// TwinCAT 3 PLC project Untitled1
// ProgramVersion: 3.1.4026.15
// libraries:
//   Tc2_Standard, * (Beckhoff Automation GmbH)
//   Tc2_System, * (Beckhoff Automation GmbH)
//   Tc2_TcpIp, * (Beckhoff Automation GmbH)
// project tree:
//   DUTs/ E_TcpIpErrorID.TcDUT, E_TcpIpState.TcDUT
//   / PlcTask.TcTTO
//   POUs/ FB_TCPIPServerManager.TcPOU, FB_TCPIPClientManager.TcPOU, MAIN.TcPOU
// real-time tasks:
//   TASK PlcTask: cycle T#10ms, priority 20, ADS port 350

CONFIGURATION Untitled1
    RESOURCE PLC ON TwinCAT3
        TASK PlcTask(INTERVAL := T#10ms, PRIORITY := 20);
        PROGRAM MAIN WITH PlcTask : MAIN;
    END_RESOURCE
END_CONFIGURATION

// ---- DUTs/E_TcpIpErrorID.TcDUT
{attribute 'qualified_only'}
//{attribute 'strict'}
{attribute 'to_string'}
TYPE E_TcpIpErrorID :
(
	ERR_NOERROR := 0,
	ERR_INTERNAL := 1,
	ERR_NORTIME := 2,
	ERR_ALLOCLOCKEDMEM := 3,
	ERR_INSERTMAILBOX := 4,
	ERR_WRONGRECEIVEHMSG := 5,
	ERR_TARGETPORTNOTFOUND := 6,
	ERR_TARGETMACHINENOTFOUND := 7,
	ERR_UNKNOWNCMDID := 8,
	ERR_BADTASKID := 9,
	ERR_NOIO := 10,
	ERR_UNKNOWNAMSCMD := 11,
	ERR_WIN32ERROR := 12,
	ERR_PORTNOTCONNECTED := 13,
	ERR_INVALIDAMSLENGTH := 14,
	ERR_INVALIDAMSNETID := 15,
	ERR_LOWINSTLEVEL := 16,
	ERR_NODEBUGINTAVAILABLE := 17,
	ERR_PORTDISABLED := 18,
	ERR_PORTALREADYCONNECTED := 19,
	ERR_AMSSYNC_W32ERROR := 20,
	ERR_AMSSYNC_TIMEOUT := 21,
	ERR_AMSSYNC_AMSERROR := 22,
	ERR_AMSSYNC_NOINDEXINMAP := 23,
	ERR_INVALIDAMSPORT := 24,
	ERR_NOMEMORY := 25,
	ERR_TCPSEND := 26,
	ERR_HOSTUNREACHABLE := 27,
	ERR_INVALIDAMSFRAGMENT := 28,
	ERR_TLSSEND := 29,
	ERR_ACCESSDENIED := 30,

	(* Router error codes *)
	ROUTERERR_NOLOCKEDMEMORY := 1280,
	ROUTERERR_RESIZEMEMORY := 1281,
	ROUTERERR_MAILBOXFULL := 1282,
	ROUTERERR_DEBUGBOXFULL := 1283,
	ROUTERERR_UNKNOWNPORTTYPE := 1284,
	ROUTERERR_NOTINITIALIZED := 1285,
	ROUTERERR_PORTALREADYINUSE := 1286,
	ROUTERERR_NOTREGISTERED := 1287,
	ROUTERERR_NOMOREQUEUES := 1288,
	ROUTERERR_INVALIDPORT := 1289,
	ROUTERERR_NOTACTIVATED := 1290,
	ROUTERERR_FRAGMENTBOXFULL := 1291,
	ROUTERERR_FRAGMENTTIMEOUT := 1292,
	ROUTERERR_TOBEREMOVED := 1293,

	(* General ADS error codes *)
	ADSERR_DEVICE_ERROR := 1792,
	ADSERR_DEVICE_SRVNOTSUPP := 1793,
	ADSERR_DEVICE_INVALIDGRP := 1794,
	ADSERR_DEVICE_INVALIDOFFSET := 1795,
	ADSERR_DEVICE_INVALIDACCESS := 1796,
	ADSERR_DEVICE_INVALIDSIZE := 1797,
	ADSERR_DEVICE_INVALIDDATA := 1798,
	ADSERR_DEVICE_NOTREADY := 1799,
	ADSERR_DEVICE_BUSY := 1800,
	ADSERR_DEVICE_INVALIDCONTEXT := 1801,
	ADSERR_DEVICE_NOMEMORY := 1802,
	ADSERR_DEVICE_INVALIDPARM := 1803,
	ADSERR_DEVICE_NOTFOUND := 1804,
	ADSERR_DEVICE_SYNTAX := 1805,
	ADSERR_DEVICE_INCOMPATIBLE := 1806,
	ADSERR_DEVICE_EXISTS := 1807,
	ADSERR_DEVICE_SYMBOLNOTFOUND := 1808,
	ADSERR_DEVICE_SYMBOLVERSIONINVALID := 1809,
	ADSERR_DEVICE_INVALIDSTATE := 1810,
	ADSERR_DEVICE_TRANSMODENOTSUPP := 1811,
	ADSERR_DEVICE_NOTIFYHNDINVALID := 1812,
	ADSERR_DEVICE_CLIENTUNKNOWN := 1813,
	ADSERR_DEVICE_NOMOREHDLS := 1814,
	ADSERR_DEVICE_INVALIDWATCHSIZE := 1815,
	ADSERR_DEVICE_NOTINIT := 1816,
	ADSERR_DEVICE_TIMEOUT := 1817,
	ADSERR_DEVICE_NOINTERFACE := 1818,
	ADSERR_DEVICE_INVALIDINTERFACE := 1819,
	ADSERR_DEVICE_INVALIDCLSID := 1820,
	ADSERR_DEVICE_INVALIDOBJID := 1821,
	ADSERR_DEVICE_PENDING := 1822,
	ADSERR_DEVICE_ABORTED := 1823,
	ADSERR_DEVICE_WARNING := 1824,
	ADSERR_DEVICE_INVALIDARRAYIDX := 1825,
	ADSERR_DEVICE_SYMBOLNOTACTIVE := 1826,
	ADSERR_DEVICE_ACCESSDENIED := 1827,
	ADSERR_DEVICE_LICENSENOTFOUND := 1828,
	ADSERR_DEVICE_LICENSEEXPIRED := 1829,
	ADSERR_DEVICE_LICENSEEXCEEDED := 1830,
	ADSERR_DEVICE_LICENSEINVALID := 1831,
	ADSERR_DEVICE_LICENSESYSTEMID := 1832,
	ADSERR_DEVICE_LICENSENOTIMELIMIT := 1833,
	ADSERR_DEVICE_LICENSEFUTUREISSUE := 1834,
	ADSERR_DEVICE_LICENSETIMETOLONG := 1835,
	ADSERR_DEVICE_EXCEPTION := 1836,
	ADSERR_DEVICE_LICENSEDUPLICATED := 1837,
	ADSERR_DEVICE_SIGNATUREINVALID := 1838,
	ADSERR_DEVICE_CERTIFICATEINVALID := 1839,
	ADSERR_DEVICE_LICENSEOEMNOTFOUND := 1840,
	ADSERR_DEVICE_LICENSERESTRICTED := 1841,
	ADSERR_DEVICE_LICENSEDEMODENIED := 1842,
	ADSERR_DEVICE_INVALIDFNCID := 1843,
	ADSERR_DEVICE_OUTOFRANGE := 1844,
	ADSERR_DEVICE_INVALIDALIGNMENT := 1845,
	ADSERR_DEVICE_LICENSEPLATFORM := 1846,
	ADSERR_DEVICE_FORWARD_PL := 1847,
	ADSERR_DEVICE_FORWARD_DL := 1848,
	ADSERR_DEVICE_FORWARD_RT := 1849,
	ADSERR_CLIENT_ERROR := 1856,
	ADSERR_CLIENT_INVALIDPARM := 1857,
	ADSERR_CLIENT_LISTEMPTY := 1858,
	ADSERR_CLIENT_VARUSED := 1859,
	ADSERR_CLIENT_DUPLINVOKEID := 1860,
	ADSERR_CLIENT_SYNCTIMEOUT := 1861,
	ADSERR_CLIENT_W32ERROR := 1862,
	ADSERR_CLIENT_TIMEOUTINVALID := 1863,
	ADSERR_CLIENT_PORTNOTOPEN := 1864,
	ADSERR_CLIENT_NOAMSADDR := 1865,
	ADSERR_CLIENT_SYNCINTERNAL := 1872,
	ADSERR_CLIENT_ADDHASH := 1873,
	ADSERR_CLIENT_REMOVEHASH := 1874,
	ADSERR_CLIENT_NOMORESYM := 1875,
	ADSERR_CLIENT_SYNCRESINVALID := 1876,
	ADSERR_CLIENT_SYNCPORTLOCKED := 1877,
    ADSERR_CLIENT_REQUESTCANCELLED := 1878,

	(* RTime error codes *)
	RTERR_INTERNAL := 4096,
	RTERR_BADTIMERPERIODS := 4097,
	RTERR_INVALIDTASKPTR := 4098,
	RTERR_INVALIDSTACKPTR := 4099,
	RTERR_PRIOEXISTS := 4100,
	RTERR_NOMORETCB := 4101,
	RTERR_NOMORESEMAS := 4102,
	RTERR_NOMOREQUEUES := 4103,
	RTERR_EXTIRQALREADYDEF := 4109,
	RTERR_EXTIRQNOTDEF := 4110,
	RTERR_EXTIRQINSTALLFAILED := 4111,
	RTERR_IRQLNOTLESSOREQUAL := 4112,
	RTERR_VMXNOTSUPPORTED := 4119,
	RTERR_VMXDISABLED := 4120,
	RTERR_VMXCONTROLSMISSING := 4121,
	RTERR_VMXENABLEFAILS := 4122,

	(* Specific positive HRESULT Return Codes *)
	(* Note: HRESULT values are converted to decimal.
	   S_OK (0) conflicts with ERR_NOERROR (0)
	   S_FALSE (1) conflicts with ERR_INTERNAL (1) *)
	S_PENDING := 515, (* 0x0203 *)
	S_WATCHDOG_TIMEOUT := 598, (* 0x0256 *)

	(* TCP Winsock error codes *)
	WSAETIMEDOUT := 10060,
	WSAECONNREFUSED := 10061,
	WSAEHOSTUNREACH := 10065
)UDINT;
END_TYPE

// ---- DUTs/E_TcpIpState.TcDUT
{attribute 'qualified_only'}
{attribute 'strict'}
{attribute 'to_string'}
TYPE E_TcpIpState :
(
	Idle := 0,
	//initSend := 9,
	Send := 10,
	//initReceive := 19,
	Receive := 20,
	Error := -1
);
END_TYPE

// ---- POUs/MAIN.TcPOU
PROGRAM MAIN
VAR CONSTANT
	DATA_SIZE : UDINT := 255;
END_VAR
VAR
	fbTcpIpManager : FB_TcpIpServerManager<DATA_SIZE>('192.168.10.160',5000);
	fbTcpIpClient :	FB_TcpIpClientManager<DATA_SIZE>('192.168.10.160',5000);
	step : INT;
	
	sSend 		: STRING(DATA_SIZE);
	sReceive 	: STRING(DATA_SIZE);
	sSend2 		: STRING(DATA_SIZE);
	sReceive2 	: STRING(DATA_SIZE);
END_VAR

CASE step OF
	0:;
	
	1:
		fbTcpIpManager.Enable();
		
		step := 0;
		
	2:
		fbTcpIpManager.Disable();
		
		step := 0;
		
	3:
		IF fbTcpIpManager.Receive(sReceive) THEN
			step := 0;
		END_IF
		
	4:
		IF fbTcpIpManager.Send(sSend) THEN
			step := 0;
		END_IF
		
		
	11:
		fbTcpIpClient.Enable();
		
		step := 0;
		
	12:
		fbTcpIpClient.Disable();
		
		step := 0;
		
	13:
		IF fbTcpIpClient.Receive(sReceive2) THEN
			step := 0;
		END_IF
		
	14:
		IF fbTcpIpClient.Send(sSend2) THEN
			step := 0;
		END_IF
		
		
END_CASE

fbTcpIpManager.CyclicCall();
fbTcpIpClient.CyclicCall();

END_PROGRAM

// ---- POUs/FB_TCPIPServerManager.TcPOU
FUNCTION_BLOCK FB_TCPIPServerManager

VAR_GENERIC CONSTANT
	STRING_SIZE 		: UDINT := 255;
END_VAR

VAR
	_Initalized : BOOL;
	fbServerClientConnection 	: FB_ServerClientConnection;
	fbSocketCloseAll			: FB_SocketCloseAll;
	fbSocketSend				: FB_SocketSend;
	fbSocketReceive				: FB_SocketReceive;
	eState 						: E_TcpIpState;
	
	_sSrvNetID 					: T_AmsNetID  := ''; 
	_LocalHost 					: T_IPv4Addr := '192.168.10.160';
	_LocalPort 					: UDINT := 5000;
	hServer 					: T_HSERVER;
	_SendString					: REFERENCE TO STRING(STRING_SIZE);
	_ReceiveString				: REFERENCE TO STRING(STRING_SIZE);
	_SendDone 					: BOOL;
	_ReceiveDone 				: BOOL;
	
	_ErrorID 	: UDINT;
	
	NumberOfSentData 		: UDINT;
	NumberOfReceivedData 	: UDINT;
END_VAR

ACTION CyclicCall:
IF NOT _Initalized THEN
	fbSocketCloseAll(sSrvNetId:= _sSrvNetID, bExecute:= NOT _Initalized);
	IF fbSocketCloseAll.bBusy THEN
		RETURN;
	ELSE
		fbSocketCloseAll(sSrvNetId:= _sSrvNetID, bExecute:= FALSE);
	END_IF
	_Initalized := F_CreateServerHnd(
	sSrvNetID := _sSrvNetID, 
	sLocalHost:= _LocalHost, 
	nLocalPort:= _LocalPort, 
	nMode     := LISTEN_MODE_CLOSEALL, 
	bEnable   := TRUE, 
	hServer   := hServer);
	eState := E_TcpIpState.Idle;
	RETURN;
END_IF

fbServerClientConnection(hServer:= hServer);
IF fbServerClientConnection.bError THEN
	eState := E_TcpIpState.Error;
END_IF 	

CASE eState OF
	E_TcpIpState.Idle:;
	
	E_TcpIpState.Send:
		fbSocketSend(sSrvNetId:= _sSrvNetID, hSocket:= fbServerClientConnection.hSocket, 
			cbLen:= STRING_SIZE, 
			pSrc:= ADR(_SendString), 
			bExecute:= TRUE);
		IF NOT fbSocketSend.bBusy THEN
			IF NumberOfSentData <  4294967290 THEN
				NumberOfSentData := NumberOfSentData + 1;
			ELSE
				NumberOfSentData := 0;
			END_IF
			eState := E_TcpIpState.Idle;
		ELSIF fbSocketSend.bError THEN
			 eState := E_TcpipState.Error;
			 _ErrorID := fbSocketSend.nErrId;
		END_IF

	E_TcpIpState.Receive:
		fbSocketReceive(sSrvNetId:= _sSrvNetID, hSocket:= fbServerClientConnection.hSocket, 
			cbLen:= STRING_SIZE, 
			pDest:= ADR(_ReceiveString), 
			bExecute:= TRUE);
		IF NOT fbSocketReceive.bBusy THEN
			eState := E_TcpipState.Idle;
			IF NumberOfReceivedData <  4294967290 THEN
				NumberOfReceivedData := NumberOfReceivedData + 1;
			ELSE
				NumberOfReceivedData := 0;
			END_IF
		ELSIF fbSocketReceive.bError THEN
			 eState := E_TcpipState.Error;
			 _ErrorID := fbSocketReceive.nErrId;
		END_IF
	
	E_TcpIpState.Error:;
	
END_CASE
END_ACTION

METHOD Disable
VAR_INPUT
END_VAR
fbServerClientConnection.bEnable := FALSE;
eState := E_TcpIpState.Idle;
END_METHOD

METHOD Enable
VAR_INPUT
END_VAR
fbServerClientConnection.bEnable := TRUE;
eState := E_TcpIpState.Idle;
END_METHOD

PROPERTY ErrorID : UDINT
GET
IF eState = E_TcpIpState.Error THEN
	ErrorID := _ErrorID;
ELSE
	ErrorID := 0;
END_IF
END_GET
END_PROPERTY

//FB_Init is always available implicitly and it is used primarily for initialization.
//The return value is not evaluated. For a specific influence, you can also declare the
//methods explicitly and provide additional code there with the standard initialization
//code. You can evaluate the return value.
METHOD FB_Init: BOOL
VAR_INPUT
    bInitRetains: BOOL; // TRUE: the retain variables are initialized (reset warm / reset cold)
    bInCopyCode: BOOL;  // TRUE: the instance will be copied to the copy code afterward (online change)   
	LocalHost 					: T_IPv4Addr := '192.168.10.160';
	LocalPort 					: UDINT := 5000;
END_VAR
_LocalHost := LocalHost;
_LocalPort := LocalPort;
END_METHOD

PROPERTY isConnected : BOOL
GET
isConnected := fbServerClientConnection.eState = eSocket_Connected;
END_GET
END_PROPERTY

PROPERTY isError : BOOL
GET
isError := eState = E_TcpIpState.Error;
END_GET
END_PROPERTY

METHOD Receive : BOOL
VAR_IN_OUT
	ReceiveString : STRING(STRING_SIZE);
END_VAR
_ReceiveDone := FALSE;
IF eState = E_TcpIpState.Idle THEN
	_ReceiveString REF= ReceiveString;	
	fbSocketReceive(bExecute:= FALSE);
	eState := E_Tcpipstate.Receive;
	MEMSET(ADR(_ReceiveString),0,SIZEOF(_ReceiveString));
	Receive := TRUE;
ELSE
	Receive := FALSE;
	RETURN;
END_IF
END_METHOD

METHOD Send : BOOL
VAR_IN_OUT
	SendString : STRING(STRING_SIZE);
END_VAR
_SendDone := FALSE;
IF eState = E_TcpIpState.Idle THEN
	_SendString REF= SendString;	
	fbSocketSend(bExecute:= FALSE);
	eState := E_Tcpipstate.Send;
	Send := TRUE;
ELSE
	Send := FALSE;
	RETURN;
END_IF
END_METHOD

METHOD SetReconnectTime
VAR_INPUT
	ReconnectTime : TIME;
END_VAR
fbServerClientConnection.tReconnect := ReconnectTime;
END_METHOD

END_FUNCTION_BLOCK

// ---- POUs/FB_TCPIPClientManager.TcPOU
FUNCTION_BLOCK FB_TCPIPClientManager

VAR_GENERIC CONSTANT
	STRING_SIZE 		: UDINT := 255;
END_VAR

VAR
	_Initalized : BOOL;
	fbClientConnection 			: FB_ClientServerConnection;
	fbSocketCloseAll			: FB_SocketCloseAll;
	fbSocketSend				: FB_SocketSend;
	fbSocketReceive				: FB_SocketReceive;
	eState 						: E_TcpIpState;
	
	_sSrvNetID 					: T_AmsNetID  := ''; 
// 	_RemoteHost 				: T_IPv4Addr := '192.168.10.160';
// 	_RemotePort 				: UDINT := 5000;
	_SendString					: REFERENCE TO STRING(STRING_SIZE);
	_ReceiveString				: REFERENCE TO STRING(STRING_SIZE);
	_SendDone 					: BOOL;
	_ReceiveDone 				: BOOL;
	
	_ErrorID 				: E_TcpIpErrorID;
	
	RTrig_SendData			: R_TRIG;
	RTrig_ReceiveData		: R_TRIG;
	NumberOfSentData 		: UDINT;
	NumberOfReceivedData 	: UDINT;
END_VAR

ACTION CyclicCall:
IF NOT _Initalized THEN
	fbSocketCloseAll(sSrvNetId:= _sSrvNetID, bExecute:= NOT _Initalized);
	IF fbSocketCloseAll.bBusy THEN
		RETURN;
	ELSE
		fbSocketCloseAll(sSrvNetId:= _sSrvNetID, bExecute:= FALSE);
		_Initalized := TRUE;
	END_IF
END_IF


fbClientConnection();
IF fbClientConnection.bError THEN
	eState := E_TcpIpState.Error;
END_IF 	


fbSocketSend(sSrvNetId:= _sSrvNetID, hSocket:= fbClientConnection.hSocket, cbLen:= STRING_SIZE, pSrc:= ADR(_SendString));
IF fbSocketSend.bError THEN
	 eState := E_TcpipState.Error;
	 _ErrorID := fbSocketSend.nErrId;
ELSIF NOT fbSocketSend.bBusy THEN
	_SendDone := TRUE;
END_IF

fbSocketReceive(sSrvNetId:= _sSrvNetID, hSocket:= fbClientConnection.hSocket, cbLen:= STRING_SIZE, pDest:= ADR(_ReceiveString));
IF fbSocketReceive.bError THEN
	 eState := E_TcpipState.Error;
	 _ErrorID := fbSocketReceive.nErrId;
ELSIF NOT fbSocketReceive.bBusy THEN
	_ReceiveDone := TRUE;
END_IF




RTrig_ReceiveData(CLK := NOT (fbSocketReceive.bBusy OR fbSocketReceive.bError));
IF RTrig_ReceiveData.Q THEN
	IF NumberOfReceivedData <  4294967290 THEN
		NumberOfReceivedData := NumberOfReceivedData + 1;
	ELSE
		NumberOfReceivedData := 0;
	END_IF	
END_IF

RTrig_SendData(CLK := NOT (fbSocketSend.bBusy OR fbSocketSend.bError));
IF RTrig_SendData.Q THEN
	IF NumberOfSentData <  4294967290 THEN
		NumberOfSentData := NumberOfSentData + 1;
	ELSE
		NumberOfSentData := 0;
	END_IF	
END_IF
END_ACTION

METHOD Disable
VAR_INPUT
END_VAR
fbClientConnection.bEnable := FALSE;
END_METHOD

METHOD Enable
VAR_INPUT
END_VAR
fbClientConnection.bEnable := TRUE;
NumberOfSentData 		:= 0;
NumberOfReceivedData 	:= 0;
END_METHOD

PROPERTY ErrorID : E_TcpIpErrorID
GET
IF eState = E_TcpIpState.Error THEN
	ErrorID := _ErrorID;
ELSE
	ErrorID := 0;
END_IF
END_GET
END_PROPERTY

//FB_Init is always available implicitly and it is used primarily for initialization.
//The return value is not evaluated. For a specific influence, you can also declare the
//methods explicitly and provide additional code there with the standard initialization
//code. You can evaluate the return value.
METHOD FB_Init: BOOL
VAR_INPUT
    bInitRetains: BOOL; // TRUE: the retain variables are initialized (reset warm / reset cold)
    bInCopyCode: BOOL;  // TRUE: the instance will be copied to the copy code afterward (online change)   
	RemoteHost 					: T_IPv4Addr := '192.168.10.160';
	RemotePort 					: UDINT := 5000;
END_VAR
fbClientConnection.sRemoteHost := RemoteHost;
fbClientConnection.nRemotePort := RemotePort;
END_METHOD

PROPERTY isConnected : BOOL
GET
isConnected := fbClientConnection.eState = eSocket_Connected;
END_GET
END_PROPERTY

PROPERTY isError : BOOL
GET
isError := eState = E_TcpIpState.Error;
END_GET
END_PROPERTY

PROPERTY isReceived : BOOL
GET
isReceived := _ReceiveDone;
END_GET
END_PROPERTY

PROPERTY isSent : BOOL
GET
isSent := _SendDone;
END_GET
END_PROPERTY

METHOD Receive : BOOL
VAR_IN_OUT
	ReceiveString : STRING(STRING_SIZE);
END_VAR
_ReceiveDone := FALSE;
IF NOT fbSocketReceive.bBusy THEN
	_ReceiveString REF= ReceiveString;	
	fbSocketReceive(bExecute:= FALSE);
	fbSocketReceive.bExecute := TRUE;
	eState := E_Tcpipstate.Receive;
	MEMSET(ADR(_ReceiveString),0,SIZEOF(_ReceiveString));
	Receive := TRUE;
ELSE
	Receive := FALSE;
	RETURN;
END_IF
END_METHOD

METHOD Send : BOOL
VAR_IN_OUT
	SendString : STRING(STRING_SIZE);
END_VAR
_SendDone := FALSE;
IF NOT fbSocketSend.bBusy THEN
	_SendString REF= SendString;	
	fbSocketSend(bExecute:= FALSE);
	fbSocketSend.bExecute := TRUE;
	eState := E_Tcpipstate.Send;
	Send := TRUE;
ELSE
	Send := FALSE;
	RETURN;
END_IF
END_METHOD

METHOD SetReconnectTime
VAR_INPUT
	ReconnectTime : TIME;
END_VAR
fbClientConnection.tReconnect := ReconnectTime;
END_METHOD

END_FUNCTION_BLOCK
